// TIA Portal V20 export
FUNCTION "CallShiftModel" : Void   // FC2, LAD
TITLE = CallShiftModel
// Called LSicar_Shiftmodel
// stored: IsIECCheckEnabled true, SetENOAutomatically true
   VAR_TEMP   // added for the SCL form of the ladder/FBD networks
      _w1 : Bool;
      _w2 : Bool;
      _w3 : Bool;
   END_VAR
BEGIN

REGION Network 1: BLOCK INFO HEADER
   // SIEMENS AG / (c)Copyright 2023
   // ------------------------------------------------------------------------------
   // Title:            CallShiftModel (FC2)
   // Comment/Function: Called LSicar_Shiftmodel 
   // Library/Family:   Automation Framework
   // Author:           Siemens Digital Industry
   // Tested with:      ---
   // Engineering:      TIA Portal V19
   // Restrictions:     -
   // Requirements:     ---
   // ------------------------------------------------------------------------------
   // Change log table:
   // Version  | Date       | Expert in charge       | Changes applied
   // ---------|------------|------------------------|------------------------------
   // 01.00.00 | 11.12.2023 | Siemens Industry Online Support
   //                         First released version
END_REGION

REGION Network 2: Call: shiftmodel
   // FB for handling the shift model and times
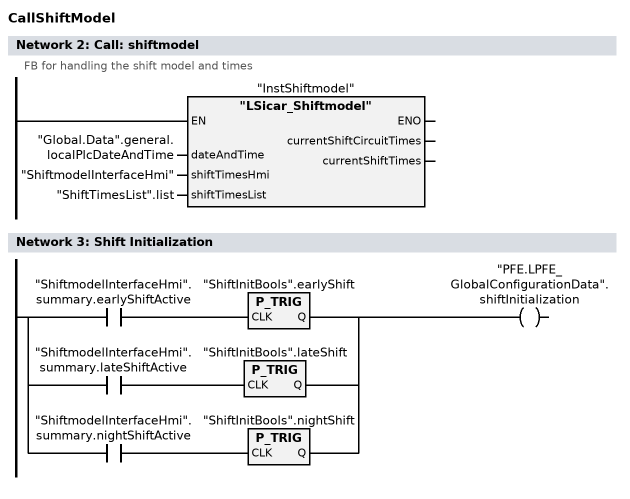
   RUNG wire#powerrail
      "InstShiftmodel"(dateAndTime := "Global.Data".general.localPlcDateAndTime, shiftTimesHmi := "ShiftmodelInterfaceHmi", shiftTimesList := "ShiftTimesList".list, currentShiftCircuitTimes =>, currentShiftTimes =>)
   END_RUNG
   // the same network as SCL:
   "InstShiftmodel"(dateAndTime := "Global.Data".general.localPlcDateAndTime,   // "LSicar_Shiftmodel"
                    shiftTimesHmi := "ShiftmodelInterfaceHmi",
                    shiftTimesList := "ShiftTimesList".list);
END_REGION

REGION Network 3: Shift Initialization
   RUNG wire#powerrail
      Contact( "ShiftmodelInterfaceHmi".summary.earlyShiftActive )
      P_Trig( "ShiftInitBools".earlyShift )
      wire#w1
      Coil( "PFE.LPFE_GlobalConfigurationData".shiftInitialization )
   END_RUNG
   RUNG wire#powerrail
      Contact( "ShiftmodelInterfaceHmi".summary.lateShiftActive )
      P_Trig( "ShiftInitBools".lateShift )
   END_RUNG wire#w1
   RUNG wire#powerrail
      Contact( "ShiftmodelInterfaceHmi".summary.nightShiftActive )
      P_Trig( "ShiftInitBools".nightShift )
   END_RUNG wire#w1
   // the same network as SCL:
   #_w1 := "ShiftmodelInterfaceHmi".summary.earlyShiftActive AND NOT "ShiftInitBools".earlyShift;   // rising edge
   "ShiftInitBools".earlyShift := "ShiftmodelInterfaceHmi".summary.earlyShiftActive;
   #_w2 := "ShiftmodelInterfaceHmi".summary.lateShiftActive AND NOT "ShiftInitBools".lateShift;   // rising edge
   "ShiftInitBools".lateShift := "ShiftmodelInterfaceHmi".summary.lateShiftActive;
   #_w3 := "ShiftmodelInterfaceHmi".summary.nightShiftActive AND NOT "ShiftInitBools".nightShift;   // rising edge
   "ShiftInitBools".nightShift := "ShiftmodelInterfaceHmi".summary.nightShiftActive;
   "PFE.LPFE_GlobalConfigurationData".shiftInitialization := #_w1 OR #_w2 OR #_w3;
END_REGION
END_FUNCTION
